(* IEC 61131-3 sources: Schneider_04_new/HMIRemote (part 2) *)

				(* Retrieving events *)
				udiev := Video_GetEvent( res );
				(* Extracting the event code *)
				ev := TO_UINT(udiev);

				CASE ev OF

				(* Key-related events handling: *)
				kWM_KEY:

					key := TO_USINT(SHR(udiev, 16));

					CASE key OF

					11:	(* Key: Up - Action: PrevField *)
						iNextSel := TO_INT( Video_PrevEdit( TRUE ) );
						IF iNextSel > -1 THEN
							res := Video_SendEvent( kWM_SELECT, TO_UINT(iNextSel) );
						END_IF;

					10:	(* Key: Down - Action: NextField *)
						iNextSel := TO_INT( Video_NextEdit( TRUE ) );
						IF iNextSel > -1 THEN
							res := Video_SendEvent( kWM_SELECT, TO_UINT(iNextSel) );
						END_IF;

					13:	(* Key: Enter - Action: Edit *)

						CASE iNextSel OF

							65:
								(* Entering the edit mode *)
								res := Video_EnterEdit( TO_UINT( iNextSel ) );

								IF res = kKEY_Up THEN

									iNextSel := TO_INT( Video_NextEdit( TRUE ) );
									IF iNextSel > -1 THEN
										res := Video_SendEvent( kWM_SELECT, TO_UINT(iNextSel) );
									END_IF;

								ELSIF res = kKEY_Down THEN

									iNextSel := TO_INT( Video_PrevEdit( TRUE ) );
									IF iNextSel > -1 THEN
										res := Video_SendEvent( kWM_SELECT, TO_UINT(iNextSel) );
									END_IF;

								END_IF;

						END_CASE;

								CASE iNextSel OF

									64:	(* Button: Button_2 - Action: OpenPage 'configureKNS' *)
									res := Video_Lock( res );
									guiCallStack[ giStackPtr ] := 8;
									RETURN;

								END_CASE;

					END_CASE;

				(* Selecting a control: *)
				kWM_SELECT:

					(* Extracting the index of the edit box clicked *)
					iNextSel := TO_INT(SHR(udiev, 16));

					(* Only select the object *)
					res := Video_EnterEditSel( TO_UINT( iNextSel ), TRUE );

					END_CASE;
				END_IF;

			END_WHILE;

		END_WHILE;

	END_FUNCTION_BLOCK

FUNCTION_BLOCK Drawlogin

	VAR_OUTPUT
	uiOutVar : UINT;
	END_VAR

	VAR_EXTERNAL
	guiCallStack : ARRAY[ 0..9 ] OF UINT;
	giStackPtr : INT;
	fbBackPage : DrawBackPage;
	login_password_1 : INT;
	login_password_2 : INT;
	login_password_3 : INT;
	login_password_4 : INT;
	login_visible_login : BOOL;
	fbloginEdit_1 : EditBox01;
	fbloginEdit_2 : EditBox01;
	fbloginEdit_3 : EditBox01;
	fbloginEdit_4 : EditBox01;
	fbloginButton_5 : Button02;
	$waitRefresh : BOOL;
	END_VAR

	VAR
	res : USINT;
	bStatRedrw : BOOL;
	bMapsReset : BOOL;
	iNextSel : INT;
	$Set_IndexVisEl : UINT;
	$Set_CycleRefresh : UINT;
	$Set_PtrBoolVis : @BOOL;
	$Set_VisEl : BOOL;
	$Set_IndexPageInSet : UINT;
	$Set_ForcePageReload : BOOL;
	$Set_NextPage : BOOL;
	$Set_PrevPage : BOOL;
	$Set_LocalSetPagNumber: UINT;
	$Set_NumVisEl: UINT;
	$Set_LastFirstEl: INT;
	udiev : UDINT;
	ev : UINT;
	key : USINT;
	x1 : UINT;
	y1 : UINT;
	x2 : UINT;
	y2 : UINT;
	wParam : UINT;
	END_VAR

	{CODE:ST}

	(* Writing this page's ID to the top of the callstack *)
	guiCallStack[ giStackPtr ] := 16#07;

	(* Manage back page index for opening page *)
	fbBackPage.IsOpening := TRUE;
	fbBackPage.CurrPageId := 16#07;
	fbBackPage();

	(* Flag of waiting for refresh task *)
	$waitRefresh := TRUE;

	(* Resetting the object map *)
	res := Video_ResetMaps( 16#00 );

	(* Setting flags: this page is to be drawn *)
	bStatRedrw := TRUE;
	bMapsReset := TRUE;

	(* The area to be cleared is the area of the entire page *)
	x1:= 0;
	y1:= 0;
	x2:= 127;
	y2:= 63;

	(* Unlocking the video *)
	res := Video_Unlock( res );

	WHILE TRUE DO

		(* Locking the video *)
		res := Video_Lock( res );

		(* Initializing the page *)
		res := Video_InitPage( 0, 0, 127, 63, ?' ', 16#0003 );

		(* Setting the page colors *)
		res := Video_SetPageColors( 0, 16777215 );

		IF bStatRedrw THEN

			(* *** CLEARING PAGE AREA *** *)
			res := Video_ClrRect( x1, y1, x2, y2 );

		END_IF;

		IF bMapsReset THEN

			(* Resetting all maps *)
			res := Video_ResetMaps( 16#FF );

			(* *** DRAW PAGE CONTROLS *** *)

			(* *** PAGE SECTION *** *)

			(* *** DRAW CONTROLS *** *)
			fbloginEdit_1.accMode := kACS_INIT;
			fbloginEdit_1();
			fbloginEdit_1.accMode := kACS_PRINT;
			(* Object: Edit_1 - Event: AfterUpdate - ProcName: check_password *)
			if login_password_1 = 1 and login_password_2 = 7 and login_password_3 = 0 and login_password_4 = 4 then login_visible_login := true ;
			end_if ;
			(* End of associated procedure *)
			fbloginEdit_2.accMode := kACS_INIT;
			fbloginEdit_2();
			fbloginEdit_2.accMode := kACS_PRINT;
			(* Object: Edit_2 - Event: AfterUpdate - ProcName: check_password *)
			if login_password_1 = 1 and login_password_2 = 7 and login_password_3 = 0 and login_password_4 = 4 then login_visible_login := true ;
			end_if ;
			(* End of associated procedure *)
			fbloginEdit_3.accMode := kACS_INIT;
			fbloginEdit_3();
			fbloginEdit_3.accMode := kACS_PRINT;
			(* Object: Edit_3 - Event: AfterUpdate - ProcName: check_password *)
			if login_password_1 = 1 and login_password_2 = 7 and login_password_3 = 0 and login_password_4 = 4 then login_visible_login := true ;
			end_if ;
			(* End of associated procedure *)
			fbloginEdit_4.accMode := kACS_INIT;
			fbloginEdit_4();
			fbloginEdit_4.accMode := kACS_PRINT;
			(* Object: Edit_4 - Event: AfterUpdate - ProcName: check_password *)
			if login_password_1 = 1 and login_password_2 = 7 and login_password_3 = 0 and login_password_4 = 4 then login_visible_login := true ;
			end_if ;
			(* End of associated procedure *)
			fbloginButton_5.accMode := kACS_INIT;
			fbloginButton_5();
			fbloginButton_5.accMode := kACS_PRINT;

			(* Select the first selectable control *)
			iNextSel := Video_FirstLastEdit( TRUE, FALSE );
			IF iNextSel > -1 THEN
				res := Video_SendEvent( kWM_SELECT, TO_UINT(iNextSel) );
			END_IF;

		END_IF;

		(* Unlocking the video *)
		res := Video_Unlock( res );

		(* Reset the flags for page redraw request *)
		bStatRedrw := FALSE;
		bMapsReset := FALSE;

		(* *** EVENTS HANDLING *** *)
		WHILE TRUE DO

			(* the drawing task wait the refreshing task *)
			IF $waitRefresh THEN
				res := Video_Sleep( 50 );
			ELSE

				(* Retrieving events *)
				udiev := Video_GetEvent( res );
				(* Extracting the event code *)
				ev := TO_UINT(udiev);

				CASE ev OF

				(* Key-related events handling: *)
				kWM_KEY:

					key := TO_USINT(SHR(udiev, 16));

					CASE key OF

					8:	(* Key: Left - Action: OpenPage *)
					res := Video_Lock( res );
					guiCallStack[ giStackPtr ] := 0;
					RETURN;

					11:	(* Key: Up - Action: PrevField *)
						iNextSel := TO_INT( Video_PrevEdit( TRUE ) );
						IF iNextSel > -1 THEN
							res := Video_SendEvent( kWM_SELECT, TO_UINT(iNextSel) );
						END_IF;

					10:	(* Key: Down - Action: NextField *)
						iNextSel := TO_INT( Video_NextEdit( TRUE ) );
						IF iNextSel > -1 THEN
							res := Video_SendEvent( kWM_SELECT, TO_UINT(iNextSel) );
						END_IF;

					13:	(* Key: Enter - Action: Edit *)

						CASE iNextSel OF

							67,68,69,70:
								(* Entering the edit mode *)
								res := Video_EnterEdit( TO_UINT( iNextSel ) );

								IF res = kKEY_Up THEN

									iNextSel := TO_INT( Video_NextEdit( TRUE ) );
									IF iNextSel > -1 THEN
										res := Video_SendEvent( kWM_SELECT, TO_UINT(iNextSel) );
									END_IF;

								ELSIF res = kKEY_Down THEN

									iNextSel := TO_INT( Video_PrevEdit( TRUE ) );
									IF iNextSel > -1 THEN
										res := Video_SendEvent( kWM_SELECT, TO_UINT(iNextSel) );
									END_IF;

								END_IF;

						END_CASE;

								CASE iNextSel OF
									66:	(* Object: Button_5 - Event: OnPress - ProcName: reset_login *)
									login_visible_login := false ;
									login_password_1 := 0 ;
									login_password_2 := 0 ;
									login_password_3 := 0 ;
									login_password_4 := 0 ;
									(* End of associated procedure *)

								END_CASE;

								CASE iNextSel OF

									66:	(* Button: Button_5 - Action: OpenPage 'menu' *)
									res := Video_Lock( res );
									guiCallStack[ giStackPtr ] := 4;
									RETURN;

								END_CASE;

					END_CASE;

				(* Selecting a control: *)
				kWM_SELECT:

					(* Extracting the index of the edit box clicked *)
					iNextSel := TO_INT(SHR(udiev, 16));

					(* Only select the object *)
					res := Video_EnterEditSel( TO_UINT( iNextSel ), TRUE );

					END_CASE;
				END_IF;

			END_WHILE;

		END_WHILE;

	END_FUNCTION_BLOCK

FUNCTION_BLOCK DrawconfigureKNS

	VAR_OUTPUT
	uiOutVar : UINT;
	END_VAR

	VAR_EXTERNAL
	guiCallStack : ARRAY[ 0..9 ] OF UINT;
	giStackPtr : INT;
	fbBackPage : DrawBackPage;
	fbconfigureKNSButton_1 : Button02;
	fbconfigureKNSButton_2 : Button02;
	fbconfigureKNSButton_3 : Button02;
	fbconfigureKNSButton_4 : Button02;
	fbconfigureKNSButton_5 : Button02;
	$waitRefresh : BOOL;
	END_VAR

	VAR
	res : USINT;
	bStatRedrw : BOOL;
	bMapsReset : BOOL;
	iNextSel : INT;
	$Set_IndexVisEl : UINT;
	$Set_CycleRefresh : UINT;
	$Set_PtrBoolVis : @BOOL;
	$Set_VisEl : BOOL;
	$Set_IndexPageInSet : UINT;
	$Set_ForcePageReload : BOOL;
	$Set_NextPage : BOOL;
	$Set_PrevPage : BOOL;
	$Set_LocalSetPagNumber: UINT;
	$Set_NumVisEl: UINT;
	$Set_LastFirstEl: INT;
	udiev : UDINT;
	ev : UINT;
	key : USINT;
	x1 : UINT;
	y1 : UINT;
	x2 : UINT;
	y2 : UINT;
	wParam : UINT;
	END_VAR

	{CODE:ST}

	(* Writing this page's ID to the top of the callstack *)
	guiCallStack[ giStackPtr ] := 16#08;

	(* Manage back page index for opening page *)
	fbBackPage.IsOpening := TRUE;
	fbBackPage.CurrPageId := 16#08;
	fbBackPage();

	(* Flag of waiting for refresh task *)
	$waitRefresh := TRUE;

	(* Resetting the object map *)
	res := Video_ResetMaps( 16#00 );

	(* Setting flags: this page is to be drawn *)
	bStatRedrw := TRUE;
	bMapsReset := TRUE;

	(* The area to be cleared is the area of the entire page *)
	x1:= 0;
	y1:= 0;
	x2:= 127;
	y2:= 63;

	(* Unlocking the video *)
	res := Video_Unlock( res );

	WHILE TRUE DO

		(* Locking the video *)
		res := Video_Lock( res );

		(* Initializing the page *)
		res := Video_InitPage( 0, 0, 127, 63, ?' ', 16#0003 );

		(* Setting the page colors *)
		res := Video_SetPageColors( 0, 16777215 );

		IF bStatRedrw THEN

			(* *** CLEARING PAGE AREA *** *)
			res := Video_ClrRect( x1, y1, x2, y2 );

		END_IF;

		IF bMapsReset THEN

			(* Resetting all maps *)
			res := Video_ResetMaps( 16#FF );

			(* *** DRAW PAGE CONTROLS *** *)

			(* *** PAGE SECTION *** *)

			(* *** DRAW CONTROLS *** *)
			fbconfigureKNSButton_1.accMode := kACS_INIT;
			fbconfigureKNSButton_1();
			fbconfigureKNSButton_1.accMode := kACS_PRINT;
			fbconfigureKNSButton_2.accMode := kACS_INIT;
			fbconfigureKNSButton_2();
			fbconfigureKNSButton_2.accMode := kACS_PRINT;
			fbconfigureKNSButton_3.accMode := kACS_INIT;
			fbconfigureKNSButton_3();
			fbconfigureKNSButton_3.accMode := kACS_PRINT;
			fbconfigureKNSButton_4.accMode := kACS_INIT;
			fbconfigureKNSButton_4();
			fbconfigureKNSButton_4.accMode := kACS_PRINT;
			fbconfigureKNSButton_5.accMode := kACS_INIT;
			fbconfigureKNSButton_5();
			fbconfigureKNSButton_5.accMode := kACS_PRINT;

			(* Select the first selectable control *)
			iNextSel := Video_FirstLastEdit( TRUE, FALSE );
			IF iNextSel > -1 THEN
				res := Video_SendEvent( kWM_SELECT, TO_UINT(iNextSel) );
			END_IF;

		END_IF;

		(* Unlocking the video *)
		res := Video_Unlock( res );

		(* Reset the flags for page redraw request *)
		bStatRedrw := FALSE;
		bMapsReset := FALSE;

		(* *** EVENTS HANDLING *** *)
		WHILE TRUE DO

			(* the drawing task wait the refreshing task *)
			IF $waitRefresh THEN
				res := Video_Sleep( 50 );
			ELSE

				(* Retrieving events *)
				udiev := Video_GetEvent( res );
				(* Extracting the event code *)
				ev := TO_UINT(udiev);

				CASE ev OF

				(* Key-related events handling: *)
				kWM_KEY:

					key := TO_USINT(SHR(udiev, 16));

					CASE key OF

					11:	(* Key: Up - Action: PrevField *)
						iNextSel := TO_INT( Video_PrevEdit( TRUE ) );
						IF iNextSel > -1 THEN
							res := Video_SendEvent( kWM_SELECT, TO_UINT(iNextSel) );
						END_IF;

					10:	(* Key: Down - Action: NextField *)
						iNextSel := TO_INT( Video_NextEdit( TRUE ) );
						IF iNextSel > -1 THEN
							res := Video_SendEvent( kWM_SELECT, TO_UINT(iNextSel) );
						END_IF;

					13:	(* Key: Enter - Action: Edit *)

								CASE iNextSel OF

									71:	(* Button: Button_1 - Action: OpenPage 'updateRotation' *)
									res := Video_Lock( res );
									guiCallStack[ giStackPtr ] := 1;
									RETURN;

									72:	(* Button: Button_2 - Action: OpenPage 'updateLVL' *)
									res := Video_Lock( res );
									guiCallStack[ giStackPtr ] := 5;
									RETURN;

									73:	(* Button: Button_3 - Action: OpenPage 'resetAlarmPumps' *)
									res := Video_Lock( res );
									guiCallStack[ giStackPtr ] := 6;
									RETURN;

									74:	(* Button: Button_4 - Action: OpenPage 'pumpsPriority' *)
									res := Video_Lock( res );
									guiCallStack[ giStackPtr ] := 9;
									RETURN;

									75:	(* Button: Button_5 - Action: OpenPage 'menu' *)
									res := Video_Lock( res );
									guiCallStack[ giStackPtr ] := 4;
									RETURN;

								END_CASE;

					END_CASE;

				(* Selecting a control: *)
				kWM_SELECT:

					(* Extracting the index of the edit box clicked *)
					iNextSel := TO_INT(SHR(udiev, 16));

					(* Only select the object *)
					res := Video_EnterEditSel( TO_UINT( iNextSel ), TRUE );

					END_CASE;
				END_IF;

			END_WHILE;

		END_WHILE;

	END_FUNCTION_BLOCK

FUNCTION_BLOCK DrawpumpsPriority

	VAR_OUTPUT
	uiOutVar : UINT;
	END_VAR

	VAR_EXTERNAL
	guiCallStack : ARRAY[ 0..9 ] OF UINT;
	giStackPtr : INT;
	fbBackPage : DrawBackPage;
	fbpumpsPriorityString_4 : Static01;
	fbpumpsPriorityString_5 : Static01;
	fbpumpsPriorityString_6 : Static01;
	fbpumpsPriorityEdit_1 : EditBox01;
	fbpumpsPriorityEdit_2 : EditBox01;
	fbpumpsPriorityEdit_3 : EditBox01;
	fbpumpsPriorityButton_7 : Button02;
	fbParampumpsPriority : ParampumpsPriority;
	$waitRefresh : BOOL;
	END_VAR

	VAR
	res : USINT;
	bStatRedrw : BOOL;
	bMapsReset : BOOL;
	iNextSel : INT;
	$Set_IndexVisEl : UINT;
	$Set_CycleRefresh : UINT;
	$Set_PtrBoolVis : @BOOL;
	$Set_VisEl : BOOL;
	$Set_IndexPageInSet : UINT;
	$Set_ForcePageReload : BOOL;
	$Set_NextPage : BOOL;
	$Set_PrevPage : BOOL;
	$Set_LocalSetPagNumber: UINT;
	$Set_NumVisEl: UINT;
	$Set_LastFirstEl: INT;
	udiev : UDINT;
	ev : UINT;
	key : USINT;
	x1 : UINT;
	y1 : UINT;
	x2 : UINT;
	y2 : UINT;
	wParam : UINT;
	END_VAR

	{CODE:ST}

	(* Writing this page's ID to the top of the callstack *)
	guiCallStack[ giStackPtr ] := 16#09;

	(* Manage back page index for opening page *)
	fbBackPage.IsOpening := TRUE;
	fbBackPage.CurrPageId := 16#09;
	fbBackPage();

	(* Flag of waiting for refresh task *)
	$waitRefresh := TRUE;

	(* Resetting the object map *)
	res := Video_ResetMaps( 16#00 );

	(* Setting flags: this page is to be drawn *)
	bStatRedrw := TRUE;
	bMapsReset := TRUE;

	(* The area to be cleared is the area of the entire page *)
	x1:= 0;
	y1:= 13;
	x2:= 127;
	y2:= 63;

	(* Unlocking the video *)
	res := Video_Unlock( res );

	WHILE TRUE DO

		(* Locking the video *)
		res := Video_Lock( res );

		(* Initializing the page *)
		res := Video_InitPage( 0, 0, 127, 63, ?'$D0$9F$D1$80i$D0$BE$D1$80$D0$B8$D1$82$D0$B5$D1$82$D0$B8 $D0$BD$D0$B0$D1$81$D0$BE$D1$81i$D0$B2', 16#0103 );

		(* Setting the page colors *)
		res := Video_SetPageColors( 0, 16777215 );

		IF bStatRedrw THEN

			(* *** CLEARING PAGE AREA *** *)
			res := Video_ClrRect( x1, y1, x2, y2 );

		END_IF;

		IF bMapsReset THEN

			(* Resetting all maps *)
			res := Video_ResetMaps( 16#FF );

			(* *** OBTAIN PARAMETER VALUES *** *)
			fbParampumpsPriority();

			(* *** DRAW PAGE CONTROLS *** *)

			(* *** PAGE SECTION *** *)

			(* *** DRAW CONTROLS *** *)
			fbpumpsPriorityEdit_1.accMode := kACS_INIT;
			fbpumpsPriorityEdit_1();
			fbpumpsPriorityEdit_1.accMode := kACS_PRINT;
			fbpumpsPriorityEdit_2.accMode := kACS_INIT;
			fbpumpsPriorityEdit_2();
			fbpumpsPriorityEdit_2.accMode := kACS_PRINT;
			fbpumpsPriorityEdit_3.accMode := kACS_INIT;
			fbpumpsPriorityEdit_3();
			fbpumpsPriorityEdit_3.accMode := kACS_PRINT;
			fbpumpsPriorityString_4.accMode := kACS_INIT;
			fbpumpsPriorityString_4();
			fbpumpsPriorityString_4.accMode := kACS_PRINT;
			fbpumpsPriorityString_5.accMode := kACS_INIT;
			fbpumpsPriorityString_5();
			fbpumpsPriorityString_5.accMode := kACS_PRINT;
			fbpumpsPriorityString_6.accMode := kACS_INIT;
			fbpumpsPriorityString_6();
			fbpumpsPriorityString_6.accMode := kACS_PRINT;
			fbpumpsPriorityButton_7.accMode := kACS_INIT;
			fbpumpsPriorityButton_7();
			fbpumpsPriorityButton_7.accMode := kACS_PRINT;

			(* Select the first selectable control *)
			iNextSel := Video_FirstLastEdit( TRUE, FALSE );
			IF iNextSel > -1 THEN
				res := Video_SendEvent( kWM_SELECT, TO_UINT(iNextSel) );
			END_IF;

		END_IF;

		(* Unlocking the video *)
		res := Video_Unlock( res );

		(* Reset the flags for page redraw request *)
		bStatRedrw := FALSE;
		bMapsReset := FALSE;

		(* *** EVENTS HANDLING *** *)
		WHILE TRUE DO

			(* the drawing task wait the refreshing task *)
			IF $waitRefresh THEN
				res := Video_Sleep( 50 );
			ELSE

				(* Retrieving events *)
				udiev := Video_GetEvent( res );
				(* Extracting the event code *)
				ev := TO_UINT(udiev);

				CASE ev OF

				(* Key-related events handling: *)
				kWM_KEY:

					key := TO_USINT(SHR(udiev, 16));

					CASE key OF

					11:	(* Key: Up - Action: PrevField *)
						iNextSel := TO_INT( Video_PrevEdit( TRUE ) );
						IF iNextSel > -1 THEN
							res := Video_SendEvent( kWM_SELECT, TO_UINT(iNextSel) );
						END_IF;

					10:	(* Key: Down - Action: NextField *)
						iNextSel := TO_INT( Video_NextEdit( TRUE ) );
						IF iNextSel > -1 THEN
							res := Video_SendEvent( kWM_SELECT, TO_UINT(iNextSel) );
						END_IF;

					13:	(* Key: Enter - Action: Edit *)

						CASE iNextSel OF

							80,81,82:
								(* Entering the edit mode *)
								res := Video_EnterEdit( TO_UINT( iNextSel ) );

								IF res = kKEY_Up THEN

									iNextSel := TO_INT( Video_NextEdit( TRUE ) );
									IF iNextSel > -1 THEN
										res := Video_SendEvent( kWM_SELECT, TO_UINT(iNextSel) );
									END_IF;

								ELSIF res = kKEY_Down THEN

									iNextSel := TO_INT( Video_PrevEdit( TRUE ) );
									IF iNextSel > -1 THEN
										res := Video_SendEvent( kWM_SELECT, TO_UINT(iNextSel) );
									END_IF;

								END_IF;

						END_CASE;

								CASE iNextSel OF

									79:	(* Button: Button_7 - Action: OpenPage 'configureKNS' *)
									res := Video_Lock( res );
									guiCallStack[ giStackPtr ] := 8;
									RETURN;

								END_CASE;

					END_CASE;

				(* Selecting a control: *)
				kWM_SELECT:

					(* Extracting the index of the edit box clicked *)
					iNextSel := TO_INT(SHR(udiev, 16));

					(* Only select the object *)
					res := Video_EnterEditSel( TO_UINT( iNextSel ), TRUE );

					END_CASE;
				END_IF;

			END_WHILE;

		END_WHILE;

	END_FUNCTION_BLOCK

	(***************************)
	(*                         *)
	(* REFRESHING FUN. BLOCKS  *)
	(*                         *)
	(***************************)

FUNCTION_BLOCK Refrmain

	VAR_EXTERNAL
	guiCallStack : ARRAY[ 0..9 ] OF UINT;
	giStackPtr : INT;
	fbmainString_6 : Static01;
	fbmainString_7 : Static01;
	fbmainString_8 : Static01;
	fbmainString_22 : Static01;
	fbmainString_24 : Static01;
	fbmainEdit_2 : EditBox01;
	fbmainEdit_3 : EditBox01;
	fbmainEdit_4 : EditBox01;
	fbmainEdit_5 : EditBox01;
	fbmainEdit_10 : EditBox01;
	fbmainEdit_11 : EditBox01;
	fbmainEdit_12 : EditBox01;
	fbmainEdit_23 : EditBox01;
	fbmainEdit_25 : EditBox01;
	fbmainProgress_1 : Progress;
	fbParammain : Parammain;
	$waitRefresh : BOOL;
	END_VAR

	VAR
	res : USINT;
	pagID : UINT;
	n : USINT;
	iSP : INT;
	pDC : UDINT;
	rx1 : UINT;
	ry1 : UINT;
	rx2 : UINT;
	ry2 : UINT;
	END_VAR

	{CODE:ST}

	REPEAT

		(* Locking the video *)
		res := Video_Lock( res );

		(* Testing if page has changed *)
		pagID := guiCallStack[ giStackPtr ];

		IF pagID = 16#00 THEN

			(* the refresh task is arrived *)
			$waitRefresh := FALSE;

			(* *** REFRESH PARAMETERS *** *)
			fbParammain();

			(* *** REFRESH PAGE CONTROLS *** *)
			fbmainProgress_1();
			fbmainEdit_2();
			fbmainEdit_3();
			fbmainEdit_4();
			fbmainEdit_5();
			fbmainEdit_10();
			fbmainEdit_11();
			fbmainEdit_12();
			fbmainEdit_23();
			fbmainEdit_25();

			(* *** REFRESHING BACKGROUND ITEMS *** *)
			(* Cursor across the call stack *)
			iSP := giStackPtr;

			(* *** REFRESHING PARENT BACKGROUND ITEMS *** *)

		END_IF;

		(* Unlocking the video *)
		res := Video_Unlock( res );

		(* Suspending the task *)
		res := Video_Sleep( 50 );

	UNTIL pagID <> 16#00
	END_REPEAT;

END_FUNCTION_BLOCK

FUNCTION_BLOCK RefrupdateRotation

	VAR_EXTERNAL
	guiCallStack : ARRAY[ 0..9 ] OF UINT;
	giStackPtr : INT;
	fbupdateRotationEdit_2 : EditBox01;
	fbupdateRotationButton_5 : Button02;
	$waitRefresh : BOOL;
	END_VAR

	VAR
	res : USINT;
	pagID : UINT;
	n : USINT;
	iSP : INT;
	pDC : UDINT;
	rx1 : UINT;
	ry1 : UINT;
	rx2 : UINT;
	ry2 : UINT;
	END_VAR

	{CODE:ST}

	REPEAT

		(* Locking the video *)
		res := Video_Lock( res );

		(* Testing if page has changed *)
		pagID := guiCallStack[ giStackPtr ];

		IF pagID = 16#01 THEN

			(* the refresh task is arrived *)
			$waitRefresh := FALSE;

			(* *** REFRESH PAGE CONTROLS *** *)
			IF fbupdateRotationEdit_2.accMode <> kACS_MODIFY THEN
				fbupdateRotationEdit_2();
			END_IF;

			(* *** REFRESHING BACKGROUND ITEMS *** *)
			(* Cursor across the call stack *)
			iSP := giStackPtr;

			(* *** REFRESHING PARENT BACKGROUND ITEMS *** *)

		END_IF;

		(* Unlocking the video *)
		res := Video_Unlock( res );

		(* Suspending the task *)
		res := Video_Sleep( 50 );

	UNTIL pagID <> 16#01
	END_REPEAT;

END_FUNCTION_BLOCK

FUNCTION_BLOCK RefrSetupRS2

	VAR_EXTERNAL
	guiCallStack : ARRAY[ 0..9 ] OF UINT;
	giStackPtr : INT;
	fbSetupRS2String_1 : Static01;
	fbSetupRS2String_2 : Static01;
	fbSetupRS2String_3 : Static01;
	fbSetupRS2String_4 : Static01;
	fbSetupRS2String_5 : Static01;
	fbSetupRS2String_6 : Static01;
	fbSetupRS2Edit_7 : EditBox01;
	fbSetupRS2Edit_8 : EditBox01;
	fbSetupRS2Edit_9 : EditBox01;
	fbSetupRS2Edit_10 : EditBox01;
	fbSetupRS2Edit_11 : EditBox01;
	fbSetupRS2Edit_12 : EditBox01;
	$waitRefresh : BOOL;
	END_VAR

	VAR
	res : USINT;
	pagID : UINT;
	n : USINT;
	iSP : INT;
	pDC : UDINT;
	rx1 : UINT;
	ry1 : UINT;
	rx2 : UINT;
	ry2 : UINT;
	END_VAR

	{CODE:ST}

	REPEAT

		(* Locking the video *)
		res := Video_Lock( res );

		(* Testing if page has changed *)
		pagID := guiCallStack[ giStackPtr ];

		IF pagID = 16#02 THEN

			(* the refresh task is arrived *)
			$waitRefresh := FALSE;

			(* *** REFRESH PAGE CONTROLS *** *)
			IF fbSetupRS2Edit_7.accMode <> kACS_MODIFY THEN
				fbSetupRS2Edit_7();
			END_IF;
			IF fbSetupRS2Edit_8.accMode <> kACS_MODIFY THEN
				fbSetupRS2Edit_8();
			END_IF;
			IF fbSetupRS2Edit_9.accMode <> kACS_MODIFY THEN
				fbSetupRS2Edit_9();
			END_IF;
			IF fbSetupRS2Edit_10.accMode <> kACS_MODIFY THEN
				fbSetupRS2Edit_10();
			END_IF;
			IF fbSetupRS2Edit_11.accMode <> kACS_MODIFY THEN
				fbSetupRS2Edit_11();
			END_IF;
			IF fbSetupRS2Edit_12.accMode <> kACS_MODIFY THEN
				fbSetupRS2Edit_12();
			END_IF;

			(* *** REFRESHING BACKGROUND ITEMS *** *)
			(* Cursor across the call stack *)
			iSP := giStackPtr;

			(* *** REFRESHING PARENT BACKGROUND ITEMS *** *)

		END_IF;

		(* Unlocking the video *)
		res := Video_Unlock( res );

		(* Suspending the task *)
		res := Video_Sleep( 50 );

	UNTIL pagID <> 16#02
	END_REPEAT;

END_FUNCTION_BLOCK

FUNCTION_BLOCK RefrSetupIP

	VAR_EXTERNAL
	guiCallStack : ARRAY[ 0..9 ] OF UINT;
	giStackPtr : INT;
	fbSetupIPString_1 : Static01;
	fbSetupIPString_2 : Static01;
	fbSetupIPString_3 : Static01;
	fbSetupIPString_4 : Static01;
	fbSetupIPEdit_5 : EditBox01;
	fbSetupIPEdit_6 : EditBox01;
	fbSetupIPEdit_7 : EditBox01;
	fbSetupIPEdit_8 : EditBox01;
	fbSetupIPEdit_9 : EditBox01;
	fbSetupIPEdit_10 : EditBox01;
	fbSetupIPEdit_11 : EditBox01;
	fbSetupIPEdit_12 : EditBox01;
	fbSetupIPEdit_13 : EditBox01;
	fbSetupIPEdit_14 : EditBox01;
	fbSetupIPEdit_15 : EditBox01;
	fbSetupIPEdit_16 : EditBox01;
	fbSetupIPEdit_17 : EditBox01;
	fbSetupIPEdit_18 : EditBox01;
	fbSetupIPEdit_19 : EditBox01;
	fbSetupIPEdit_20 : EditBox01;
	$waitRefresh : BOOL;
	END_VAR

	VAR
	res : USINT;
	pagID : UINT;
	n : USINT;
	iSP : INT;
	pDC : UDINT;
	rx1 : UINT;
	ry1 : UINT;
	rx2 : UINT;
	ry2 : UINT;
	END_VAR

	{CODE:ST}

	REPEAT

		(* Locking the video *)
		res := Video_Lock( res );

		(* Testing if page has changed *)
		pagID := guiCallStack[ giStackPtr ];

		IF pagID = 16#03 THEN

			(* the refresh task is arrived *)
			$waitRefresh := FALSE;

			(* *** REFRESH PAGE CONTROLS *** *)
			IF fbSetupIPEdit_5.accMode <> kACS_MODIFY THEN
				fbSetupIPEdit_5();
			END_IF;
			IF fbSetupIPEdit_6.accMode <> kACS_MODIFY THEN
				fbSetupIPEdit_6();
			END_IF;
			IF fbSetupIPEdit_7.accMode <> kACS_MODIFY THEN
				fbSetupIPEdit_7();
			END_IF;
			IF fbSetupIPEdit_8.accMode <> kACS_MODIFY THEN
				fbSetupIPEdit_8();
			END_IF;
			IF fbSetupIPEdit_9.accMode <> kACS_MODIFY THEN
				fbSetupIPEdit_9();
			END_IF;
			IF fbSetupIPEdit_10.accMode <> kACS_MODIFY THEN
				fbSetupIPEdit_10();
			END_IF;
			IF fbSetupIPEdit_11.accMode <> kACS_MODIFY THEN
				fbSetupIPEdit_11();
			END_IF;
			IF fbSetupIPEdit_12.accMode <> kACS_MODIFY THEN
				fbSetupIPEdit_12();
			END_IF;
			IF fbSetupIPEdit_13.accMode <> kACS_MODIFY THEN
				fbSetupIPEdit_13();
			END_IF;
			IF fbSetupIPEdit_14.accMode <> kACS_MODIFY THEN
				fbSetupIPEdit_14();
			END_IF;
			IF fbSetupIPEdit_15.accMode <> kACS_MODIFY THEN
				fbSetupIPEdit_15();
			END_IF;
			IF fbSetupIPEdit_16.accMode <> kACS_MODIFY THEN
				fbSetupIPEdit_16();
			END_IF;
			IF fbSetupIPEdit_17.accMode <> kACS_MODIFY THEN
				fbSetupIPEdit_17();
			END_IF;
			IF fbSetupIPEdit_18.accMode <> kACS_MODIFY THEN
				fbSetupIPEdit_18();
			END_IF;
			IF fbSetupIPEdit_19.accMode <> kACS_MODIFY THEN
				fbSetupIPEdit_19();
			END_IF;
			IF fbSetupIPEdit_20.accMode <> kACS_MODIFY THEN
				fbSetupIPEdit_20();
			END_IF;

			(* *** REFRESHING BACKGROUND ITEMS *** *)
			(* Cursor across the call stack *)
			iSP := giStackPtr;

			(* *** REFRESHING PARENT BACKGROUND ITEMS *** *)

		END_IF;

		(* Unlocking the video *)
		res := Video_Unlock( res );

		(* Suspending the task *)
		res := Video_Sleep( 50 );

	UNTIL pagID <> 16#03
	END_REPEAT;

END_FUNCTION_BLOCK

FUNCTION_BLOCK Refrmenu

	VAR_EXTERNAL
	guiCallStack : ARRAY[ 0..9 ] OF UINT;
	giStackPtr : INT;
	fbmenuButton_2 : Button02;
	fbmenuButton_3 : Button02;
	fbmenuButton_4 : Button02;
	$waitRefresh : BOOL;
	END_VAR

	VAR
	res : USINT;
	pagID : UINT;
	n : USINT;
	iSP : INT;
	pDC : UDINT;
	rx1 : UINT;
	ry1 : UINT;
	rx2 : UINT;
	ry2 : UINT;
	END_VAR

	{CODE:ST}

	REPEAT

		(* Locking the video *)
		res := Video_Lock( res );

		(* Testing if page has changed *)
		pagID := guiCallStack[ giStackPtr ];

		IF pagID = 16#04 THEN

			(* the refresh task is arrived *)
			$waitRefresh := FALSE;

			(* *** REFRESH PAGE CONTROLS *** *)

			(* *** REFRESHING BACKGROUND ITEMS *** *)
			(* Cursor across the call stack *)
			iSP := giStackPtr;

			(* *** REFRESHING PARENT BACKGROUND ITEMS *** *)

		END_IF;

		(* Unlocking the video *)
		res := Video_Unlock( res );

		(* Suspending the task *)
		res := Video_Sleep( 50 );

	UNTIL pagID <> 16#04
	END_REPEAT;

END_FUNCTION_BLOCK

FUNCTION_BLOCK RefrupdateLVL

	VAR_EXTERNAL
	guiCallStack : ARRAY[ 0..9 ] OF UINT;
	giStackPtr : INT;
	fbupdateLVLString_1 : Static01;
	fbupdateLVLString_2 : Static01;
	fbupdateLVLString_4 : Static01;
	fbupdateLVLString_7 : Static01;
	fbupdateLVLString_10 : Static01;
	fbupdateLVLString_12 : Static01;
	fbupdateLVLString_13 : Static01;
	fbupdateLVLString_14 : Static01;
	fbupdateLVLEdit_3 : EditBox01;
	fbupdateLVLEdit_5 : EditBox01;
	fbupdateLVLEdit_8 : EditBox01;
	fbupdateLVLEdit_11 : EditBox01;
	fbParamupdateLVL : ParamupdateLVL;
	$waitRefresh : BOOL;
	END_VAR

	VAR
	res : USINT;
	pagID : UINT;
	n : USINT;
	iSP : INT;
	pDC : UDINT;
	rx1 : UINT;
	ry1 : UINT;
	rx2 : UINT;
	ry2 : UINT;
	END_VAR

	{CODE:ST}

	REPEAT

		(* Locking the video *)
		res := Video_Lock( res );

		(* Testing if page has changed *)
		pagID := guiCallStack[ giStackPtr ];

		IF pagID = 16#05 THEN

			(* the refresh task is arrived *)
			$waitRefresh := FALSE;

			(* *** REFRESH PARAMETERS *** *)
			fbParamupdateLVL();

			(* *** REFRESH PAGE CONTROLS *** *)
			IF fbupdateLVLEdit_3.accMode <> kACS_MODIFY THEN
				fbupdateLVLEdit_3();
			END_IF;
			IF fbupdateLVLEdit_5.accMode <> kACS_MODIFY THEN
				fbupdateLVLEdit_5();
			END_IF;
			IF fbupdateLVLEdit_8.accMode <> kACS_MODIFY THEN
				fbupdateLVLEdit_8();
			END_IF;
			IF fbupdateLVLEdit_11.accMode <> kACS_MODIFY THEN
				fbupdateLVLEdit_11();
			END_IF;

			(* *** REFRESHING BACKGROUND ITEMS *** *)
			(* Cursor across the call stack *)
			iSP := giStackPtr;

			(* *** REFRESHING PARENT BACKGROUND ITEMS *** *)

		END_IF;

		(* Unlocking the video *)
		res := Video_Unlock( res );

		(* Suspending the task *)
		res := Video_Sleep( 50 );

	UNTIL pagID <> 16#05
	END_REPEAT;

END_FUNCTION_BLOCK

FUNCTION_BLOCK RefrresetAlarmPumps

	VAR_EXTERNAL
	guiCallStack : ARRAY[ 0..9 ] OF UINT;
	giStackPtr : INT;
	fbresetAlarmPumpsEdit_1 : EditBox01;
	fbresetAlarmPumpsButton_2 : Button02;
	$waitRefresh : BOOL;
	END_VAR

	VAR
	res : USINT;
	pagID : UINT;
	n : USINT;
	iSP : INT;
	pDC : UDINT;
	rx1 : UINT;
	ry1 : UINT;
	rx2 : UINT;
	ry2 : UINT;
	END_VAR

	{CODE:ST}

	REPEAT

		(* Locking the video *)
		res := Video_Lock( res );

		(* Testing if page has changed *)
		pagID := guiCallStack[ giStackPtr ];

		IF pagID = 16#06 THEN

			(* the refresh task is arrived *)
			$waitRefresh := FALSE;

			(* *** REFRESH PAGE CONTROLS *** *)
			IF fbresetAlarmPumpsEdit_1.accMode <> kACS_MODIFY THEN
				fbresetAlarmPumpsEdit_1();
			END_IF;

			(* *** REFRESHING BACKGROUND ITEMS *** *)
			(* Cursor across the call stack *)
			iSP := giStackPtr;

			(* *** REFRESHING PARENT BACKGROUND ITEMS *** *)

		END_IF;

		(* Unlocking the video *)
		res := Video_Unlock( res );

		(* Suspending the task *)
		res := Video_Sleep( 50 );

	UNTIL pagID <> 16#06
	END_REPEAT;

END_FUNCTION_BLOCK

FUNCTION_BLOCK Refrlogin

	VAR_EXTERNAL
	guiCallStack : ARRAY[ 0..9 ] OF UINT;
	giStackPtr : INT;
	login_visible_login : BOOL;
	login_password_1 : INT;
	login_password_2 : INT;
	login_password_3 : INT;
	login_password_4 : INT;
	fbloginEdit_1 : EditBox01;
	fbloginEdit_2 : EditBox01;
	fbloginEdit_3 : EditBox01;
	fbloginEdit_4 : EditBox01;
	fbloginButton_5 : Button02;
	$waitRefresh : BOOL;
	END_VAR

	VAR
	res : USINT;
	pagID : UINT;
	n : USINT;
	iSP : INT;
	pDC : UDINT;
	rx1 : UINT;
	ry1 : UINT;
	rx2 : UINT;
	ry2 : UINT;
	END_VAR

	{CODE:ST}

	REPEAT

		(* Locking the video *)
		res := Video_Lock( res );

		(* Testing if page has changed *)
		pagID := guiCallStack[ giStackPtr ];

		IF pagID = 16#07 THEN

			(* the refresh task is arrived *)
			$waitRefresh := FALSE;

			(* *** REFRESH PAGE CONTROLS *** *)
			IF fbloginEdit_1.accMode <> kACS_MODIFY THEN
				fbloginEdit_1();
				(* Object: Edit_1 - Event: AfterUpdate - ProcName: check_password *)
				if login_password_1 = 1 and login_password_2 = 7 and login_password_3 = 0 and login_password_4 = 4 then login_visible_login := true ;
				end_if ;
				(* End of associated procedure *)
			END_IF;
			IF fbloginEdit_2.accMode <> kACS_MODIFY THEN
				fbloginEdit_2();
				(* Object: Edit_2 - Event: AfterUpdate - ProcName: check_password *)
				if login_password_1 = 1 and login_password_2 = 7 and login_password_3 = 0 and login_password_4 = 4 then login_visible_login := true ;
				end_if ;
				(* End of associated procedure *)
			END_IF;
			IF fbloginEdit_3.accMode <> kACS_MODIFY THEN
				fbloginEdit_3();
				(* Object: Edit_3 - Event: AfterUpdate - ProcName: check_password *)
				if login_password_1 = 1 and login_password_2 = 7 and login_password_3 = 0 and login_password_4 = 4 then login_visible_login := true ;
				end_if ;
				(* End of associated procedure *)
			END_IF;
			IF fbloginEdit_4.accMode <> kACS_MODIFY THEN
				fbloginEdit_4();
				(* Object: Edit_4 - Event: AfterUpdate - ProcName: check_password *)
				if login_password_1 = 1 and login_password_2 = 7 and login_password_3 = 0 and login_password_4 = 4 then login_visible_login := true ;
				end_if ;
				(* End of associated procedure *)
			END_IF;
			fbloginButton_5();

			(* *** REFRESHING BACKGROUND ITEMS *** *)
			(* Cursor across the call stack *)
			iSP := giStackPtr;

			(* *** REFRESHING PARENT BACKGROUND ITEMS *** *)

		END_IF;

		(* Unlocking the video *)
		res := Video_Unlock( res );

		(* Suspending the task *)
		res := Video_Sleep( 50 );

	UNTIL pagID <> 16#07
	END_REPEAT;

END_FUNCTION_BLOCK

FUNCTION_BLOCK RefrconfigureKNS

	VAR_EXTERNAL
	guiCallStack : ARRAY[ 0..9 ] OF UINT;
	giStackPtr : INT;
	fbconfigureKNSButton_1 : Button02;
	fbconfigureKNSButton_2 : Button02;
	fbconfigureKNSButton_3 : Button02;
	fbconfigureKNSButton_4 : Button02;
	fbconfigureKNSButton_5 : Button02;
	$waitRefresh : BOOL;
	END_VAR

	VAR
	res : USINT;
	pagID : UINT;
	n : USINT;
	iSP : INT;
	pDC : UDINT;
	rx1 : UINT;
	ry1 : UINT;
	rx2 : UINT;
	ry2 : UINT;
	END_VAR

	{CODE:ST}

	REPEAT

		(* Locking the video *)
		res := Video_Lock( res );

		(* Testing if page has changed *)
		pagID := guiCallStack[ giStackPtr ];

		IF pagID = 16#08 THEN

			(* the refresh task is arrived *)
			$waitRefresh := FALSE;

			(* *** REFRESH PAGE CONTROLS *** *)

			(* *** REFRESHING BACKGROUND ITEMS *** *)
			(* Cursor across the call stack *)
			iSP := giStackPtr;

			(* *** REFRESHING PARENT BACKGROUND ITEMS *** *)

		END_IF;

		(* Unlocking the video *)
		res := Video_Unlock( res );

		(* Suspending the task *)
		res := Video_Sleep( 50 );

	UNTIL pagID <> 16#08
	END_REPEAT;

END_FUNCTION_BLOCK

FUNCTION_BLOCK RefrpumpsPriority

	VAR_EXTERNAL
	guiCallStack : ARRAY[ 0..9 ] OF UINT;
	giStackPtr : INT;
	fbpumpsPriorityString_4 : Static01;
	fbpumpsPriorityString_5 : Static01;
	fbpumpsPriorityString_6 : Static01;
	fbpumpsPriorityEdit_1 : EditBox01;
	fbpumpsPriorityEdit_2 : EditBox01;
	fbpumpsPriorityEdit_3 : EditBox01;
	fbpumpsPriorityButton_7 : Button02;
	fbParampumpsPriority : ParampumpsPriority;
	$waitRefresh : BOOL;
	END_VAR

	VAR
	res : USINT;
	pagID : UINT;
	n : USINT;
	iSP : INT;
	pDC : UDINT;
	rx1 : UINT;
	ry1 : UINT;
	rx2 : UINT;
	ry2 : UINT;
	END_VAR

	{CODE:ST}

	REPEAT

		(* Locking the video *)
		res := Video_Lock( res );

		(* Testing if page has changed *)
		pagID := guiCallStack[ giStackPtr ];

		IF pagID = 16#09 THEN

			(* the refresh task is arrived *)
			$waitRefresh := FALSE;

			(* *** REFRESH PARAMETERS *** *)
			fbParampumpsPriority();

			(* *** REFRESH PAGE CONTROLS *** *)
			IF fbpumpsPriorityEdit_1.accMode <> kACS_MODIFY THEN
				fbpumpsPriorityEdit_1();
			END_IF;
			IF fbpumpsPriorityEdit_2.accMode <> kACS_MODIFY THEN
				fbpumpsPriorityEdit_2();
			END_IF;
			IF fbpumpsPriorityEdit_3.accMode <> kACS_MODIFY THEN
				fbpumpsPriorityEdit_3();
			END_IF;

			(* *** REFRESHING BACKGROUND ITEMS *** *)
			(* Cursor across the call stack *)
			iSP := giStackPtr;

			(* *** REFRESHING PARENT BACKGROUND ITEMS *** *)

		END_IF;

		(* Unlocking the video *)
		res := Video_Unlock( res );

		(* Suspending the task *)
		res := Video_Sleep( 50 );

	UNTIL pagID <> 16#09
	END_REPEAT;

END_FUNCTION_BLOCK

	(***************************)
	(*                         *)
	(* PARAMETER  FUN. BLOCKS  *)
	(*                         *)
	(***************************)

FUNCTION_BLOCK Parammain

	VAR_EXTERNAL
$Param_0_9057_0 : BOOL;
	END_VAR

	VAR
		idx : UINT;
		res : UINT;
		errorRes : ARRAY[ 0..1 ] OF UINT;
	END_VAR

	{CODE:ST}
	(* Reading parameter @LocalParameters.is_three_pumps_here *)
	errorRes[0] := Video_GetParam( 0, 9057, 0, ?$Param_0_9057_0, tyBool );

	FOR idx := 0 TO 0 DO
		(* Sending an error message if necessary *)
		IF errorRes[idx] = kPAR_ERR_NOTFOUND OR errorRes[idx] = kPAR_ERR_INVTYPE THEN
			res := Video_SendEvent( kWM_MSG, kPAR_MSG_NOTFOUND );
			EXIT;
		ELSIF errorRes[idx] <> kPAR_ERR_OK THEN
			res := Video_SendEvent( kWM_MSG, kPAR_MSG_SYSERR );
			EXIT;
		END_IF;

	END_FOR;

	END_FUNCTION_BLOCK

FUNCTION_BLOCK ParamupdateLVL

	VAR_EXTERNAL
	$Param_0_9057_0 : BOOL;
	END_VAR

	VAR
		idx : UINT;
		res : UINT;
		errorRes : ARRAY[ 0..1 ] OF UINT;
	END_VAR

	{CODE:ST}
		(* Reading parameter @LocalParameters.is_three_pumps_here *)
		errorRes[0] := Video_GetParam( 0, 9057, 0, ?$Param_0_9057_0, tyBool );

	FOR idx := 0 TO 0 DO
		(* Sending an error message if necessary *)
		IF errorRes[idx] = kPAR_ERR_NOTFOUND OR errorRes[idx] = kPAR_ERR_INVTYPE THEN
			res := Video_SendEvent( kWM_MSG, kPAR_MSG_NOTFOUND );
			EXIT;
		ELSIF errorRes[idx] <> kPAR_ERR_OK THEN
			res := Video_SendEvent( kWM_MSG, kPAR_MSG_SYSERR );
			EXIT;
		END_IF;

	END_FOR;

	END_FUNCTION_BLOCK

FUNCTION_BLOCK ParampumpsPriority

	VAR_EXTERNAL
	$Param_0_9057_0 : BOOL;
	END_VAR

	VAR
		idx : UINT;
		res : UINT;
		errorRes : ARRAY[ 0..1 ] OF UINT;
	END_VAR

	{CODE:ST}
		(* Reading parameter @LocalParameters.is_three_pumps_here *)
		errorRes[0] := Video_GetParam( 0, 9057, 0, ?$Param_0_9057_0, tyBool );

	FOR idx := 0 TO 0 DO
		(* Sending an error message if necessary *)
		IF errorRes[idx] = kPAR_ERR_NOTFOUND OR errorRes[idx] = kPAR_ERR_INVTYPE THEN
			res := Video_SendEvent( kWM_MSG, kPAR_MSG_NOTFOUND );
			EXIT;
		ELSIF errorRes[idx] <> kPAR_ERR_OK THEN
			res := Video_SendEvent( kWM_MSG, kPAR_MSG_SYSERR );
			EXIT;
		END_IF;

	END_FOR;

	END_FUNCTION_BLOCK

	(***************************)
	(*                         *)
	(*   PROC FUNCTIONS        *)
	(*                         *)
	(***************************)

FUNCTION $proc_login_check_password : BOOL

        VAR_EXTERNAL
login_password_1 : INT;
login_password_2 : INT;
login_password_3 : INT;
login_password_4 : INT;
login_visible_login : BOOL;
	END_VAR

	{ CODE:ST }
if login_password_1 = 1 and login_password_2 = 7 and login_password_3 = 0 and login_password_4 = 4 then login_visible_login := true ;
end_if ;

$proc_login_check_password:=TRUE;
END_FUNCTION

FUNCTION $proc_login_reset_login : BOOL

        VAR_EXTERNAL
login_visible_login : BOOL;
login_password_1 : INT;
login_password_2 : INT;
login_password_3 : INT;
login_password_4 : INT;
	END_VAR

	{ CODE:ST }
login_visible_login := false ;
login_password_1 := 0 ;
login_password_2 := 0 ;
login_password_3 := 0 ;
login_password_4 := 0 ;

$proc_login_reset_login:=TRUE;
END_FUNCTION
